PROGRAM Main
VAR
	//Konfiguration
	Dummy : BOOL := FALSE; //True wenn Dummy laufen soll. FALSE wenn Programm laufen soll
	
	
	//Weltframe
	pSollPose : POINTER TO RobotSollPose;
	SollPose : RobotSollPose;
	
	allIstPosArray : ARRAY[1..8] OF RobotPose;
	IstPoseCamera : RobotPose;				//kommt von der Kamera, geht zum Beobachter
	IstPoseCameraOhne0 : RobotPose;			//Nur als Plotvariable
	IstPose : RobotPose;					//kommt von Beobachter, Die offizielle IstPose
	
	//Roboframe
	SollVelo : RobotPose;
	IstVeloKlemme :RobotPose;

	IstVeloEnc : RobotPose;					//kommt von Wheelencoders, geht zu Beobachter
	
	//Bumper
	Bumperaktiv : BOOL;
	
	// Zu Gripper 
	GripperSollClose : BOOL := 0;
	GripperIstClose : BOOL := 0;
	GripperSliderAusgeloest : BOOL := 0;
	GripperLSAusgeloest : BOOL := 0;
	
	StationIstConnected : BOOL;
END_VAR

//Nur zum Plotten
IF	istPoseCamera.x <> 0 THEN
IstPoseCameraOhne0 := IstPoseCamera;
END_IF

METHOD absToDynTheta : LREAL
VAR_INPUT
	absolutThetaSoll : LREAL;
	absolutThetaIst : LREAL;
END_VAR

VAR_OUTPUT
	dynamicThetaSoll : LREAL;
END_VAR

VAR CONSTANT
	PI : LREAL := 3.1415;
END_VAR
VAR
	dTheta: LREAL;
END_VAR
(* Konvertiert einen sollTheta Wert -Pi bis - PI in einen +2Pi bis - 2Pi abhängig von der Distanz.
	So dreht sich der Robitino immer zum Kürzeren Drehwinkel in richtung Sollwinkel *) 

dTheta := absolutThetaSoll - absolutThetaIst;

IF dTheta > PI  THEN
	absToDynTheta := dTheta - 2*PI;
	
ELSIF dTheta < -PI THEN
	absToDynTheta := dTheta + 2*PI;
	
ELSE
	absToDynTheta := dTheta;
END_IF
RETURN;
END_METHOD

METHOD closeGripper : BOOL
VAR_INPUT
END_VAR
GripperSollClose := TRUE;
END_METHOD

METHOD getBumperAktiv : BOOL
VAR_INPUT
END_VAR
getBumperaktiv := Bumperaktiv;
END_METHOD

METHOD getGripperistClosed : BOOL
VAR_INPUT
END_VAR
getGripperistClosed := GripperIstClose;
END_METHOD

METHOD getGripperLSAusgeloest : BOOL
VAR_INPUT
END_VAR
getGripperLSAusgeloest := GripperLSAusgeloest;
END_METHOD

METHOD getGripperSliderAusgeloest : BOOL
VAR_INPUT
END_VAR
getGripperSliderAusgeloest := GripperSliderAusgeloest;
END_METHOD

METHOD getGripperSollClose : BOOL
VAR_INPUT
END_VAR
getGripperSollClose := GripperSollClose;
END_METHOD

METHOD getIstPose : RobotPose
VAR_INPUT
END_VAR
getIstPose := IstPose;
END_METHOD

METHOD getIstPoseCamera : RobotPose
VAR_INPUT
END_VAR
getIstPoseCamera := IstPoseCamera;
END_METHOD

METHOD getIstVeloEnc : RobotPose
VAR_INPUT
END_VAR
getIstVeloEnc := istVeloEnc;
END_METHOD

METHOD getSollPose : RobotSollPose
VAR_INPUT
END_VAR
getSollPose := SollPose;
END_METHOD

METHOD getSollVelo : RobotPose

VAR
	
END_VAR
getSollVelo:=SollVelo;
RETURN;
END_METHOD

METHOD getStationIstConnected : BOOL
VAR_INPUT
END_VAR
getStationIstConnected := StationIstConnected;
END_METHOD

METHOD istStillstand : BOOL
VAR_INPUT
END_VAR
IF SollPose.m = 0 THEN
	istStillstand := 1;
ELSE
	istStillstand := 0;
END_IF
END_METHOD

METHOD nextSollPose : BOOL
VAR_INPUT
END_VAR
IF SollPose.y <> 0 THEN
	pSollPose := pSollPose + SIZEOF(RobotSollPose);
	SollPose := pSollPose^;
END_IF
END_METHOD

METHOD openGripper : BOOL
VAR_INPUT
END_VAR
GripperSollClose := FALSE;
END_METHOD

METHOD setBumperAktiv : BOOL
VAR_INPUT
	input : BOOL;
END_VAR
Bumperaktiv := input;
END_METHOD

METHOD SetGripper : BOOL
VAR_INPUT
	status : BOOL;
END_VAR
GripperSollClose:= status;
END_METHOD

METHOD setGripperIstClosed : BOOL
VAR_INPUT
	GripperClosed : BOOL;
END_VAR
GripperIstClose := GripperClosed;
END_METHOD

METHOD setGripperLSAusgeloest : BOOL
VAR_INPUT
	input : BOOL;
END_VAR
GripperLSAusgeloest := input;
END_METHOD

METHOD setGripperSliderAusgeloest : BOOL
VAR_INPUT
	Input : BOOL; //True wenn endlage erreicht, False wenn nicht
END_VAR
GripperSliderAusgeloest := input;
END_METHOD

METHOD SetGripperSollClose : BOOL
VAR_INPUT
	input : BOOL;
END_VAR
GripperSollClose := input;
END_METHOD

METHOD setIstPose : BOOL
VAR_INPUT
	newIstPose : RobotPose;
END_VAR
IF newIstPose.y <> 0 THEN
	istPose := newIstPose;
END_IF
END_METHOD

METHOD setIstPoseCamera : BOOL
VAR_INPUT
	PoseArray : ARRAY[1..8] OF RobotPose;
END_VAR
(* Liest die richtige Kameraposition Position des Roboters aus
*)

allIstPosArray := PoseArray;
IstPoseCamera := PoseArray[Var_HAWIno.Robot_Number];

setIstPoseCamera := 1;	//Rückgabe, dass das Zuweisen erfolgreich war
RETURN;
END_METHOD

METHOD SetistVelo : BOOL
VAR_INPUT
	input : RobotPose;
END_VAR
IstVeloKlemme:=input;
END_METHOD

METHOD setIstVeloEnc : BOOL
VAR_INPUT
	IstVelo : RobotPose;
END_VAR
IstVeloEnc := IstVelo;
END_METHOD

METHOD setSollPoseArray : BOOL
VAR_INPUT
	pSollPoseArray : POINTER TO RobotSollPose;
END_VAR
pSollPose := pSollPoseArray;
SollPose := pSollPose^;
END_METHOD

METHOD SetSollVelo : Bool
VAR_INPUT
	InputVelo: RobotPose;
END_VAR

VAR
	
END_VAR
SollVelo := InputVelo;
RETURN;
END_METHOD

METHOD setStationIstConnected : BOOL
VAR_INPUT
	input : BOOL;
END_VAR
StationIstConnected := input;
END_METHOD

METHOD updateSollPose : BOOL
VAR_INPUT
END_VAR
pSollPose := pSollPose + SIZEOF(RobotSollPose);
SollPose := pSollPose^;
END_METHOD

END_PROGRAM

(* stored: Version 1.1.0.1, ProductVersion 3.1.4024.11
   POU Main: Id {000539c9-06b7-4317-a60e-77c5894f0e72}, SpecialFunc None
   Method absToDynTheta: Id {63370cd3-f23f-4ee5-9f79-7d0a25804bbc}
   Method closeGripper: Id {e0bf2792-67a9-4408-9a4f-981b57420d3c}
   Method getBumperAktiv: Id {1569796a-3828-4df0-aeda-e56ab0bc03ab}
   Method getGripperistClosed: Id {422a386d-d5e2-4c49-90cc-36b960df4459}
   Method getGripperLSAusgeloest: Id {4a372f8a-6901-466d-8544-3dc3deef8426}
   Method getGripperSliderAusgeloest: Id {b10a26e1-3b91-4eb0-84b0-ca3f3e848c55}
   Method getGripperSollClose: Id {4a8a3c33-362a-42b4-89c0-960e6b822ac6}
   Method getIstPose: Id {661b8689-a214-4bf1-87c2-c70b7fb3e145}
   Method getIstPoseCamera: Id {aaa0b453-77e2-4ce4-a7e3-020dee4d72f4}
   Method getIstVeloEnc: Id {9b6b5688-1aff-4260-8ff1-19db53a14642}
   Method getSollPose: Id {ca75675e-82ba-4b4d-90de-ba69ac754013}
   Method getSollVelo: Id {a069e554-b910-4b95-a12b-1d59a30cbeb5}
   Method getStationIstConnected: Id {17808e20-ca79-4886-8584-a65623236247}
   Method istStillstand: Id {401b72c9-ea8c-4db3-bd42-77b7d3a7597f}
   Method nextSollPose: Id {9e88087a-0a54-4a0c-a592-d5d22d0d7a48}
   Method openGripper: Id {f8476f2d-43eb-4732-8c09-57e053050d6e}
   Method setBumperAktiv: Id {0a32ea89-81ba-4373-b455-1b66a5f8c0f8}
   Method SetGripper: Id {fe0f517d-d527-4187-8760-b4f46fb6aab1}
   Method setGripperIstClosed: Id {a54c014a-0b35-42be-9f80-a414c01d1f29}
   Method setGripperLSAusgeloest: Id {a7b8d1a0-1e61-49f9-a350-a1c50ceae4d0}
   Method setGripperSliderAusgeloest: Id {20a14388-00ea-4362-88d3-7afda8f1c0b9}
   Method SetGripperSollClose: Id {89689b6c-3f0e-421f-99e9-d54b108164d4}
   Method setIstPose: Id {35c534dc-15db-433b-adbd-8a5e40f0c4b7}
   Method setIstPoseCamera: Id {965a365e-e5ba-41fa-b424-e31d8007661d}
   Method SetistVelo: Id {c106ac3b-a4cd-43f3-80b0-34c0546bad11}
   Method setIstVeloEnc: Id {b83dbb20-fe50-4129-b7a4-3ed4862ce075}
   Method setSollPoseArray: Id {4df809eb-bfb4-46d2-ab04-35704d80b4f3}
   Method SetSollVelo: Id {92ef6d32-950a-4633-9000-9da030801acf}
   Method setStationIstConnected: Id {3a38c6c0-6cf8-46c5-8f63-fb22ddb8b930}
   Method updateSollPose: Id {4e64fbed-6474-48d8-a0a4-1b1ccab63133} *)
